TYPE (* A Structured Data Type Representing a Matrix of REAL *)
  (* Standard: 61499-2 *)
  (* Version 0.0, 2002-03-05, JHC, Rockwell Automation *)
  (* Compiler header: package fb.datatype; *)
  (* Compiler Java IBM VisualAge 3.0 *)
  (* ASN.1 tag APPLICATION 23 *)
  MATRIX : STRUCT
    M : UINT; (* Number of Rows *)
    N : UINT; (* Number of Columns *)
    DATA : ARRAY [0..-1] OF REAL; (* The actual matrix,total elements=M*N as initialized *)
  END_STRUCT;
END_TYPE
